PROGRAM Axis02_Manual
VAR
//System_Bit
	Always_ON	:	BOOL	:=TRUE	;//상시 ON 
	Always_OFF	:	BOOL	:=FALSE	;//상시 OFF
END_VAR
VAR // added by the converter: edge detectors and wires of the graphical bodies
    _rt1, _rt2, _rt3, _rt4 : R_TRIG;
END_VAR

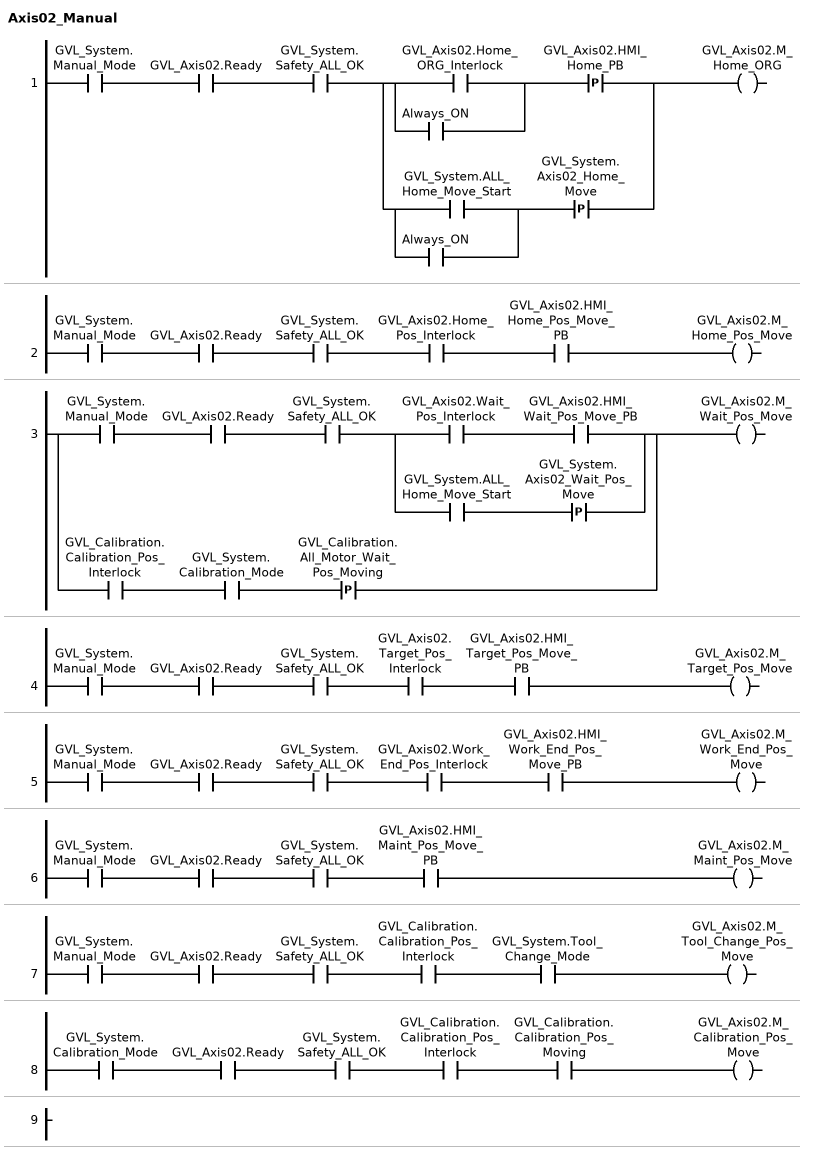
// NETWORK 1
_rt1(CLK := GVL_Axis02.HMI_Home_PB);
_rt2(CLK := GVL_System.Axis02_Home_Move);
GVL_Axis02.M_Home_ORG := GVL_System.Manual_Mode AND GVL_Axis02.Ready AND GVL_System.Safety_ALL_OK AND ((GVL_Axis02.Home_ORG_Interlock OR Always_ON) AND _rt1.Q OR (GVL_System.ALL_Home_Move_Start OR Always_ON) AND _rt2.Q);

// NETWORK 2
GVL_Axis02.M_Home_Pos_Move := GVL_System.Manual_Mode AND GVL_Axis02.Ready AND GVL_System.Safety_ALL_OK AND GVL_Axis02.Home_Pos_Interlock AND GVL_Axis02.HMI_Home_Pos_Move_PB;

// NETWORK 3
_rt3(CLK := GVL_System.Axis02_Wait_Pos_Move);
_rt4(CLK := GVL_Calibration.All_Motor_Wait_Pos_Moving);
GVL_Axis02.M_Wait_Pos_Move := GVL_System.Manual_Mode AND GVL_Axis02.Ready AND GVL_System.Safety_ALL_OK AND (GVL_Axis02.Wait_Pos_Interlock AND GVL_Axis02.HMI_Wait_Pos_Move_PB OR GVL_System.ALL_Home_Move_Start AND _rt3.Q) OR GVL_Calibration.Calibration_Pos_Interlock AND GVL_System.Calibration_Mode AND _rt4.Q;

// NETWORK 4
GVL_Axis02.M_Target_Pos_Move := GVL_System.Manual_Mode AND GVL_Axis02.Ready AND GVL_System.Safety_ALL_OK AND GVL_Axis02.Target_Pos_Interlock AND GVL_Axis02.HMI_Target_Pos_Move_PB;

// NETWORK 5
GVL_Axis02.M_Work_End_Pos_Move := GVL_System.Manual_Mode AND GVL_Axis02.Ready AND GVL_System.Safety_ALL_OK AND GVL_Axis02.Work_End_Pos_Interlock AND GVL_Axis02.HMI_Work_End_Pos_Move_PB;

// NETWORK 6
GVL_Axis02.M_Maint_Pos_Move := GVL_System.Manual_Mode AND GVL_Axis02.Ready AND GVL_System.Safety_ALL_OK AND GVL_Axis02.HMI_Maint_Pos_Move_PB;

// NETWORK 7
GVL_Axis02.M_Tool_Change_Pos_Move := GVL_System.Manual_Mode AND GVL_Axis02.Ready AND GVL_System.Safety_ALL_OK AND GVL_Calibration.Calibration_Pos_Interlock AND GVL_System.Tool_Change_Mode;

// NETWORK 8
GVL_Axis02.M_Calibration_Pos_Move := GVL_System.Calibration_Mode AND GVL_Axis02.Ready AND GVL_System.Safety_ALL_OK AND GVL_Calibration.Calibration_Pos_Interlock AND GVL_Calibration.Calibration_Pos_Moving;

// NETWORK 9

END_PROGRAM

(* stored: Version 1.1.0.1, ProductVersion 3.1.4024.15
   POU Axis02_Manual: Id {68991363-bfd2-4a1a-9fdb-072bbe628f74}, SpecialFunc None *)
